TEXTLIST WorkAreaLGVLetIn
  0 = 'Nop'
  1 = 'LGV Req In'
  2 = 'LGV End'
   = ''
END_TEXTLIST

(* stored: Version 1.1.0.1, ProductVersion 3.1.4024.11
   TextList WorkAreaLGVLetIn: Id {a03bdeca-2ca4-4027-886e-8b0477b150d3} *)
